// This function has been automatically generated from the project information.
{attribute 'signature_flag' := '1073741824'}
{attribute 'TcGenerated'}
{attribute 'no-analysis'}
FUNCTION F_GetCompany : WSTRING
VAR_INPUT
	
END_VAR

F_GetCompany := "BA Belgium";

END_FUNCTION

(* stored: Version 1.1.0.1
   POU F_GetCompany: Id {00d885d1-130e-43b0-addd-3385a7c721b4}, SpecialFunc None *)
